INTERFACE I_EnumDatatype EXTENDS I_UserDefinedDatatype

END_INTERFACE

(* stored: Version 1.1.0.1, ProductVersion 3.1.4024.12
   Itf I_EnumDatatype: Id {21dc63fa-54ad-0096-2dab-85791d8f40db} *)
